# EPICS substitutions: apps/mmfeuApp/Db/mmfeuslotFTT.substitutions
#
file "db/mmfeuslot.db" {
        pattern { P, C, S, PORT}
                {"B_DET_FTT_FEU", "1",  "1", "L1"}
                {"B_DET_FTT_FEU", "1",  "2", "L1"}
                {"B_DET_FTT_FEU", "2",  "1", "L1"}
                {"B_DET_FTT_FEU", "2",  "2", "L1"}
                {"B_DET_FTT_FEU", "3",  "1", "L1"}
                {"B_DET_FTT_FEU", "3",  "2", "L1"}
}
